# B&R Automation Studio project perfxxl (part 11)

#### rinse.c
```c
#ifdef _DEFAULT_INCLUDES
	#include <AsDefault.h>
#endif
/*
                             *******************
******************************* C SOURCE FILE *******************************
**                           *******************                           **
**                                                                         **
** project  : BlueFin                                                      **
** filename : RINSE.C                                                      **
** version  : 1.11                                                         **
** date     : 20.11.2007                                                   **
**                                                                         **
*****************************************************************************
** Abstract                                                                **
** ========                                                                **
** Handling of rinse functions: Circulation, refill, replenishing,         **
** monitoring Level and (optional) circulation switch                      **
**                                                                         **
** Copyright (c) 2007, Krause-Biagosch GmbH                                **
** All rights reserved.                                                    **
**                                                                         **
*****************************************************************************
VERSION HISTORY:
----------------
Version     : 1.00
Date        : 06.03.2007
Revised by  : Herbert Aden
Description : Original version, moved functionality from
              developertank task to here.

Version     : 1.10
Date        : 03.05.2007
Revised by  : Herbert Aden
Description : added delay for Level not ok error and delays for
              level switch on and off signal

Version     : 1.11
Date        : 20.11.2007
Revised by  : Herbert Aden
Description : added flow control functionality in mode "freshwater only",
              requires the sensor to be mounted in the inflow tube
*/
#define _RINSE_C_SRC

/****************************************************************************/
/**                                                                        **/
/**                           INCLUDE FILES                                **/
/**                                                                        **/
/****************************************************************************/

#include "egmglob_var.h"

/****************************************************************************/
/**                                                                        **/
/**                       DEFINITIONS AND MACROS                           **/
/**                                                                        **/
/****************************************************************************/
/* NONE */

/****************************************************************************/
/**                                                                        **/
/**                      TYPEDEFS AND STRUCTURES                           **/
/**                                                                        **/
/****************************************************************************/
/* NONE */

/****************************************************************************/
/**                                                                        **/
/**                      PROTOTYPES OF LOCAL FUNCTIONS                     **/
/**                                                                        **/
/****************************************************************************/
/* NONE */

/****************************************************************************/
/**                                                                        **/
/**                      EXPORTED VARIABLES                                **/
/**                                                                        **/
/****************************************************************************/
/* NONE */

/****************************************************************************/
/**                                                                        **/
/**                           GLOBAL VARIABLES                             **/
/**                                                                        **/
/****************************************************************************/
/*NONE*/

/****************************************************************************/
/**                                                                        **/
/**                      TASK-LOCAL VARIABLES                              **/
/**                                                                        **/
/****************************************************************************/
_LOCAL    UINT                RinseValveTime,RinseValveTimeToGo;

/****************************************************************************/
/**                                                                        **/
/**                    MODULE-LOCAL VARIABLES                              **/
/**                                                                        **/
/****************************************************************************/
static    TP_10ms_typ         RinseReplenishmentValveTimer;

static    TON_10ms_typ        RinseLevelOKTimer,RinseLevelNOTOKTimer,
                              RinseLevelErrorTimer,
                              RinsePumpStartTimer,
                              RinseFlowDelay,
                              RinseRefillTimer,
                              RinsePumpOffTimer,
                              RefillValveSafetyTimer;

static    R_TRIGtyp           RinsePumpCmdR,
                              RinseValveCmdR,
                              LevelOKR,
                              LevelNOTOKR;
static    F_TRIGtyp           RinseValveCmdF;

static    UINT                TmpValveTimeRinse;
static    BOOL                RinseRefillActive;

/****************************************************************************/
/**                                                                        **/
/**                      EXTERNAL VARIABLES                                **/
/**                                                                        **/
/****************************************************************************/
extern BOOL	Pulse_1s;

/****************************************************************************/
/**                                                                        **/
/**                          EXPORTED FUNCTIONS                            **/
/**                                                                        **/
/****************************************************************************/
void Rinse(void);

/******************************************************************************/
void Rinse(void)
{
/*Level*/
	RinseLevelOKTimer.IN = EGMRinse.TankFull;
	RinseLevelOKTimer.PT = 500; /*5 sec*/
	TON_10ms(&RinseLevelOKTimer);

	RinseLevelNOTOKTimer.IN = !EGMRinse.TankFull;
	RinseLevelNOTOKTimer.PT = 500; /*5 sec*/
	TON_10ms(&RinseLevelNOTOKTimer);

	LevelOKR.CLK = RinseLevelOKTimer.Q;
	LevelNOTOKR.CLK = RinseLevelNOTOKTimer.Q;
	R_TRIG(&LevelOKR);
	R_TRIG(&LevelNOTOKR);
	if(LevelOKR.Q)
		EGMRinse.LevelNotInRange = FALSE;
	if(LevelNOTOKR.Q)
		EGMRinse.LevelNotInRange = TRUE;

/* Fehlermeldung verzögern, erst wird automatisch befüllt */
	RinseLevelErrorTimer.IN = EGMRinse.LevelNotInRange;
	RinseLevelErrorTimer.PT = 2000; /* 20 s */
	TON_10ms(&RinseLevelErrorTimer);
	EGM_AlarmBitField[4] = (ModulStatus_DI == 1) && RinseLevelErrorTimer.Q && (EGMRinseParam.ReplenishingMode != FRESHWATERONLY);

/* REPLENISHING Rinse*/
/* a) per plate*/
	if (Pulse_1s &&(CurrentState == S_PROCESSING)&& (EGMRinseParam.ReplenishingMode == REPLPERPLATE))
	{
		TmpValveTimeRinse =
				((RinseReplenishmentPlateCounter * EGMRinseParam.ReplenishmentPerPlate) / EGMRinseParam.PumpMlPerSec)*100;
		if (TmpValveTimeRinse >= EGMRinseParam.MinPumpOnTime)
		{
			RinseReplenishmentValveTimer.IN = 1;
			RinseReplenishmentPlateCounter = 0;
		}
	}

/* b) per area*/
	if (Pulse_1s &&(CurrentState == S_PROCESSING)&& (EGMRinseParam.ReplenishingMode == REPLPERSQM))
	{
		TmpValveTimeRinse =
				((RinseReplenishmentSqmCounter * EGMRinseParam.ReplenishmentPerSqm) / EGMRinseParam.PumpMlPerSec)*100;
		if (TmpValveTimeRinse >= EGMRinseParam.MinPumpOnTime)
		{
			RinseReplenishmentValveTimer.IN = 1;
			RinseReplenishmentSqmCounter = 0;
		}
	}

	if (EGMRinse.Valve != OPEN )
		RinseValveTime = TmpValveTimeRinse;

	if (RinseReplenishmentValveTimer.IN && (EGMRinse.Valve != OPEN ))
		RinseReplenishmentValveTimer.PT = RinseValveTime;

	if (EGMRinse.Valve == OPEN )
		RinseValveTimeToGo = RinseReplenishmentValveTimer.PT - RinseReplenishmentValveTimer.ET;
	else
		RinseValveTimeToGo = 0;

	TP_10ms(&RinseReplenishmentValveTimer);
	RinseReplenishmentValveTimer.IN = 0;

	RinseValveCmdR.CLK = RinseReplenishmentValveTimer.Q;
	R_TRIG(&RinseValveCmdR);
	if (RinseValveCmdR.Q && (EGMRinseParam.ReplenishingMode != FRESHWATERONLY))
		EGMRinse.Valve = OPEN;

/* Ventil zu nach Zeit oder wenn kein Automatik Modus*/
	RinseValveCmdF.CLK = RinseReplenishmentValveTimer.Q && EGMRinse.Auto;
	F_TRIG(&RinseValveCmdF);
	if ((RinseValveCmdF.Q && (EGMRinseParam.ReplenishingMode != FRESHWATERONLY)) || !ControlVoltageOk)
	{
		EGMRinse.Valve = CLOSE;
	}

/*Refill Rinse*/
	TON_10ms(&RinseRefillTimer);
/* automatisch befüllen nur, wenn nicht ausschliesslich Frischwasser verwendet wird*/
	if (EGMRinseParam.ReplenishingMode != FRESHWATERONLY)
	{
		RinseRefillTimer.IN = !EGMRinse.LevelNotInRange;
		RinseRefillTimer.PT = 200;
/* Füllen nur wenn Automatik modus*/
		if (EGMRinse.LevelNotInRange && ControlVoltageOk && EGMRinse.Auto)
		{
			RinseRefillActive = TRUE;
			EGMRinse.Valve = OPEN;
		}
		if ((RinseRefillTimer.Q || !EGMRinse.Auto) && RinseRefillActive)
		{
			RinseRefillActive = FALSE;
			EGMRinse.Valve = CLOSE;
		}
	}
	else
	{
		RinseRefillTimer.IN = 0;
		RinseRefillActive = FALSE;
	}

/*
 * safety: if Valve is open and Tank full indicated close the valve after 10 sec
 */
	RefillValveSafetyTimer.IN = (EGMRinse.Valve == OPEN) && EGMRinse.TankFull;
	RefillValveSafetyTimer.PT = 1000; /* 10 sec */
	TON_10ms(&RefillValveSafetyTimer);

	if(RefillValveSafetyTimer.Q)
		EGMRinse.Valve = CLOSE;

/*Rinse Pump*/
	RinsePumpCmdR.CLK = EGMRinse.PumpCmd;
	R_TRIG(&RinsePumpCmdR);

/****************************************************************************/
/**                          Flow control                                  **/
/****************************************************************************/
	if(	EGMGlobalParam.UseRinseFlowControl )
	{
	/*
	 * wenn ausschliesslich Frischwasser verwendet wird,
	 * dann darf flow control nur  auf das geöffnete Ventil reagieren
	 */
		if (EGMRinseParam.ReplenishingMode == FRESHWATERONLY)
		{
		/*
		 * 20 sec nach Öffnen muss Durchfluß da sein
		 */
			RinsePumpStartTimer.IN = EGMRinse.Valve;
			RinsePumpStartTimer.PT = 2000; /* 20 sec */
			TON_10ms(&RinsePumpStartTimer);
			if( RinsePumpStartTimer.Q && !RinseFlowInput )
				EGM_AlarmBitField[36] = TRUE;
		}
		else
		{
	/*
	 * 20 sec nach Start der Pumpe muss Durchfluß da sein
	 */
			RinsePumpStartTimer.IN = EGMRinse.Pump;
			RinsePumpStartTimer.PT = 2000; /* 20 sec */
			TON_10ms(&RinsePumpStartTimer);
	/*
	 * wenn Frischwasser zugeführt wird, schaltet der Durchflußwächter ab,
	 * deshalb hier die Verriegelung des Fehlers mit dem Ventil
	 */
			RinseFlowDelay.IN = !RinseFlowInput && !EGMRinse.Valve;
			RinseFlowDelay.PT = 300; /* 3 sec */
			TON_10ms(&RinseFlowDelay);
			if( RinsePumpStartTimer.Q && RinseFlowDelay.Q )
				EGM_AlarmBitField[36] = TRUE;
		}
	}
	else
		EGM_AlarmBitField[36] = FALSE;

/* Rinse Pump
 * wenn 30 sec der Level nicht ok war wird die Pumpe abgeschaltet.
 * Sie kann durch steigende Flanke des Kommandos wieder für 30 s eingeschaltet werden
 * (für Service)
*/
	RinsePumpOffTimer.IN = EGMRinse.LevelNotInRange && !RinsePumpCmdR.Q;
	RinsePumpOffTimer.PT = 3000; /*30 sec*/
	TON_10ms(&RinsePumpOffTimer);
	if (RinsePumpOffTimer.Q || !ControlVoltageOk || EGM_AlarmBitField[36])
	{
		EGMRinse.Pump = OFF;
		EGMRinse.PumpCmd = OFF;
	}
	else
		EGMRinse.Pump = EGMRinse.PumpCmd;

}
/****************************************************************************/
/**                                                                        **/
/**                                 EOF                                    **/
/**                                                                        **/
/****************************************************************************/
```

#### gum.c
```c
#ifdef _DEFAULT_INCLUDES
	#include <AsDefault.h>
#endif
/*
                             *******************
******************************* C SOURCE FILE *******************************
**                           *******************                           **
**                                                                         **
** project  : BlueFin                                                      **
** filename : GUM.C                                                        **
** version  : 1.12                                                         **
** date     : 21.11.2007                                                   **
**                                                                         **
*****************************************************************************
** Abstract                                                                **
** ========                                                                **
** Handling of gumming functions: Circulation, monitoring Level            **
** and (optional) circulation switch                                       **
**                                                                         **
** Copyright (c) 2007, Krause-Biagosch GmbH                                **
** All rights reserved.                                                    **
**                                                                         **
*****************************************************************************
VERSION HISTORY:
----------------
Version     : 1.00
Date        : 06.03.2007
Revised by  : Herbert Aden
Description : Original version, moved functionality from
              developertank task to here.

Version     : 1.11
Date        : 16.11.2007
Revised by  : Herbert Aden
Description : added checking for gum valve output by monitoring an input

Version     : 1.12
Date        : 21.11.2007
Revised by  : Herbert Aden
Description : removed checking for gum valve output by monitoring an input
              (was for testing at Bauer only)
*/
#define _GUM_C_SRC

/****************************************************************************/
/**                                                                        **/
/**                           INCLUDE FILES                                **/
/**                                                                        **/
/****************************************************************************/

#include "egmglob_var.h"

/****************************************************************************/
/**                                                                        **/
/**                       DEFINITIONS AND MACROS                           **/
/**                                                                        **/
/****************************************************************************/
/* NONE */

/****************************************************************************/
/**                                                                        **/
/**                      TYPEDEFS AND STRUCTURES                           **/
/**                                                                        **/
/****************************************************************************/
/* NONE */

/****************************************************************************/
/**                                                                        **/
/**                      PROTOTYPES OF LOCAL FUNCTIONS                     **/
/**                                                                        **/
/****************************************************************************/
/* NONE */

/****************************************************************************/
/**                                                                        **/
/**                      EXPORTED VARIABLES                                **/
/**                                                                        **/
/****************************************************************************/
/* NONE */

/****************************************************************************/
/**                                                                        **/
/**                           GLOBAL VARIABLES                             **/
/**                                                                        **/
/****************************************************************************/
/*NONE*/

/****************************************************************************/
/**                                                                        **/
/**                      TASK-LOCAL VARIABLES                              **/
/**                                                                        **/
/****************************************************************************/
/*NONE*/

/****************************************************************************/
/**                                                                        **/
/**                    MODULE-LOCAL VARIABLES                              **/
/**                                                                        **/
/****************************************************************************/
static    TON_10ms_typ        GumLevelTimer,GumFlowingDelay;
static    TON_10ms_typ        GumPumpOffTimer,GumPumpStartTimer;

static    R_TRIGtyp           GumPumpCmdR;

/****************************************************************************/
/**                                                                        **/
/**                      EXTERNAL VARIABLES                                **/
/**                                                                        **/
/****************************************************************************/
extern BOOL	Pulse_1s;

/****************************************************************************/
/**                                                                        **/
/**                          EXPORTED FUNCTIONS                            **/
/**                                                                        **/
/****************************************************************************/
void Gum(void);
void InitGum(void);

/******************************************************************************/
void InitGum(void)
{
	return;
}

/******************************************************************************/
void Gum(void)
{

	if(!EGMGlobalParam.EnableGumSection && (MachineType != BLUEFIN_XS))
	{
		EGM_AlarmBitField[2] = FALSE;
		EGM_AlarmBitField[33] = FALSE;
		EGMGum.LevelNotInRange = FALSE;
		EGMGum.Pump = OFF;
		EGMGum.PumpCmd = OFF;
		EGMGum.Valve = OFF;
		EGMGum.RinseValve = OFF;
		return;
	}

/*Level Gum*/
	GumLevelTimer.IN = !EGMGum.TankFull;
	GumLevelTimer.PT = 200; /*2 sec*/
	TON_10ms(&GumLevelTimer);
	EGMGum.LevelNotInRange = GumLevelTimer.Q;
	EGM_AlarmBitField[2] = (ModulStatus_DI == 1) && EGMGum.LevelNotInRange;
/*Gum Pump*/
	GumPumpCmdR.CLK = EGMGum.PumpCmd;
	R_TRIG(&GumPumpCmdR);

	if(	EGMGlobalParam.UseGumFlowControl )
	{
	/* flow control starts 20 sec after pump start */
		GumPumpStartTimer.IN = EGMGum.Pump;
		GumPumpStartTimer.PT = 2000; /*20 sec*/
		TON_10ms(&GumPumpStartTimer);

	/* delay the "not flowing" error a bit */
		GumFlowingDelay.IN = !GumFC.Flowing;
		GumFlowingDelay.PT = 300; /* 3sec */
		TON_10ms(&GumFlowingDelay);

		if( GumPumpStartTimer.Q && GumFlowingDelay.Q )
		{
			EGM_AlarmBitField[33] = TRUE;
			GumFC.ResetMlFlown = TRUE;
		}
	}
	else
		EGM_AlarmBitField[33] = FALSE;

/* manual retrigger of the pump is possible, it will run for 5 sec */
	GumPumpOffTimer.IN = EGMGum.LevelNotInRange && !GumPumpCmdR.Q;
	GumPumpOffTimer.PT = 500; /*5 sec*/
	TON_10ms(&GumPumpOffTimer);
	if (GumPumpOffTimer.Q || !ControlVoltageOk || EGM_AlarmBitField[33])
	{
		EGMGum.Pump = OFF;
		EGMGum.PumpCmd = OFF;
	}
	else
		EGMGum.Pump = EGMGum.PumpCmd;

/*
 * safety: if the gum pump is running we always want the gum valve switched
 * and the Rinse valve closed
 */
	if( EGMGum.Pump )
	{
		EGMGum.Valve = ON;
		EGMGum.RinseValve = CLOSE;
	}

/*
 * safety: if gum rinse valve is switched on, then
 * we always want the gum valve to be switched off to make sure the
 * rinsing water cannot flow into the gum tank;
 * the Pump is switched off as well
 */
	if( EGMGum.RinseValve == OPEN )
	{
		EGMGum.Pump = EGMGum.PumpCmd = OFF;
		EGMGum.Valve = OFF;
	}
}
/****************************************************************************/
/**                                                                        **/
/**                                 EOF                                    **/
/**                                                                        **/
/****************************************************************************/
```

#### tanks.c
```c
#ifdef _DEFAULT_INCLUDES
	#include <AsDefault.h>
#endif
/*
                             *******************
******************************* C SOURCE FILE *******************************
**                           *******************                           **
**                                                                         **
** project  : BlueFin                                                      **
** filename : TANKS.C                                                      **
** version  : 1.10                                                         **
** date     : 09.03.2007                                                   **
**                                                                         **
*****************************************************************************
** Abstract                                                                **
** ========                                                                **
** Handling of Prewash, Rinse and Gum stations, basically just call        **
** functions of respective source files                                    **
**                                                                         **
** Copyright (c) 2007, Krause-Biagosch GmbH                                **
** All rights reserved.                                                    **
**                                                                         **
*****************************************************************************
VERSION HISTORY:
----------------
Version     : 1.00
Date        : 06.03.2007
Revised by  : Herbert Aden
Description : Original version, moved functionality from
              developertank task to here.

Version     : 1.10
Date        : 03.05.2007
Revised by  : Herbert Aden
Description : changes in rinse.c and prewash.c
*/
#define _TANKS_C_SRC

/****************************************************************************/
/**                                                                        **/
/**                           INCLUDE FILES                                **/
/**                                                                        **/
/****************************************************************************/
#include "egmglob_var.h"

/****************************************************************************/
/**                                                                        **/
/**                       DEFINITIONS AND MACROS                           **/
/**                                                                        **/
/****************************************************************************/
/* NONE */

/****************************************************************************/
/**                                                                        **/
/**                      TYPEDEFS AND STRUCTURES                           **/
/**                                                                        **/
/****************************************************************************/
/* NONE */

/****************************************************************************/
/**                                                                        **/
/**                      PROTOTYPES OF LOCAL FUNCTIONS                     **/
/**                                                                        **/
/****************************************************************************/
/* NONE */

/****************************************************************************/
/**                                                                        **/
/**                      PRTOTYPES OF EXTERNAL FUNCTIONS                   **/
/**                                                                        **/
/****************************************************************************/
extern void Prewash(void);
extern void Rinse(void);
extern void Gum(void);
extern void InitGum(void);

/****************************************************************************/
/**                                                                        **/
/**                      EXPORTED VARIABLES                                **/
/**                                                                        **/
/****************************************************************************/
/* NONE */

/****************************************************************************/
/**                                                                        **/
/**                           GLOBAL VARIABLES                             **/
/**                                                                        **/
/****************************************************************************/
/*NONE*/

/****************************************************************************/
/**                                                                        **/
/**                      TASK-LOCAL VARIABLES                              **/
/**                                                                        **/
/****************************************************************************/
/*NONE*/

/****************************************************************************/
/**                                                                        **/
/**                    MODULE-LOCAL VARIABLES                              **/
/**                                                                        **/
/****************************************************************************/
static    TON_10ms_typ        PulseTimer1;

/****************************************************************************/
/**                                                                        **/
/**                      EXPORTED VARIABLES                                **/
/**                                                                        **/
/****************************************************************************/
BOOL	Pulse_1s;

/****************************************************************************/
/**                                                                        **/
/**                          LOCAL FUNCTIONS                               **/
/**                                                                        **/
/****************************************************************************/

/****************************************************************************/
/** Init function, executed once at startup                                **/
/****************************************************************************/
_INIT void init()
{
	PulseTimer1.IN = 0;
	PulseTimer1.PT = 100;
	InitGum();
}

/****************************************************************************/
/** Cyclic function                                                        **/
/****************************************************************************/
_CYCLIC void cyclic()
{

	PulseTimer1.IN = 1;
	if(PulseTimer1.Q)
		PulseTimer1.IN = 0;
	TON_10ms(&PulseTimer1);
	Pulse_1s = PulseTimer1.Q;

	if(MachineType == BLUEFIN_XS)
	{
		Prewash();
		Rinse();
	}

	Gum();
	return;
}
/****************************************************************************/
/**                                                                        **/
/**                                 EOF                                    **/
/**                                                                        **/
/****************************************************************************/
```

### Program Logical/ping (ANSIC)

#### ping.c - Zyklischer Code
```c
#ifdef _DEFAULT_INCLUDES
	#include <AsDefault.h>
#endif
/****************************************************************************/
/*	TCP/IP Client Funktionalität 											*/
/*																			*/
/*																			*/
/*	Versionsgeschichte:														*/
/*  Version		Datum		Änderung								von		*/
/*	1.0			25.02.03	erste Implementation der				HA		*/
/*							Ping Funktion									*/
/*	1.10		26.02.03	SMTP Client								HA		*/
/*	1.11		15.10.15	SMTP Client removed						HA		*/
/*																			*/
/****************************************************************************/

/***** Include-Files: *****/
#include <bur/plc.h>
#include <bur/plctypes.h>
#include <string.h>
/* damit das switch unten funktioniert*/
#define _REPLACE_CONST
#include <AsICMP.h>
#include "glob_var.h"
#include <AsBrStr.h>

/***** Variablen-/Konstantendeklaration: *****/

#ifndef TRUE
#define TRUE				1
#endif
#ifndef FALSE
#define FALSE				0
#endif

USINT PingOK,PingError;
_LOCAL	IcmpPing_typ PingVar;
_LOCAL	UINT	PingOKInvisible,PingErrorInvisible;
_LOCAL USINT StartPing,IPAdr1,IPAdr2,IPAdr3,IPAdr4;

STRING IPAdress[16],tmp[10];
TOF_10ms_typ PingLEDOff;

void Ping(void)
{
	PingOKInvisible = !PingOK;
	PingErrorInvisible = !PingError;
	PingLEDOff.IN = StartPing;
	PingLEDOff.PT = 300;
	TOF_10ms(&PingLEDOff);
	if(!PingLEDOff.Q)
	{
		PingOK = 0;
		PingError = 0;
	}
	if(StartPing)
	{
		PingVar.enable = TRUE;			/* FUB enable */
		strcpy(IPAdress,"");
		brsitoa(IPAdr1,(UDINT) &tmp[0]);
		strcat(IPAdress,tmp);
		strcat(IPAdress,".");
		brsitoa(IPAdr2,(UDINT) &tmp[0]);
		strcat(IPAdress,tmp);
		strcat(IPAdress,".");
		brsitoa(IPAdr3,(UDINT) &tmp[0]);
		strcat(IPAdress,tmp);
		strcat(IPAdress,".");
		brsitoa(IPAdr4,(UDINT) &tmp[0]);
		strcat(IPAdress,tmp);
		PingVar.pHost = (UDINT)IPAdress;	/* IP Address of the Reciever */
		PingVar.timeout = 100;			/* Time of waiting */
		PingOK = 0;
		PingError = 0;
		IcmpPing(&PingVar);
		switch(PingVar.status)
		{
			case ERR_OK:
			{
				/* Ping OK */
				StartPing = FALSE;
				PingOK = 1;
				PingError = 0;
				/***********************/
				/* TODO: Go on working */
				/***********************/
				break;
			}
			case ERR_FUB_BUSY:
				/* Fub is already working */
				/* call again */
				break;
			case icmpERR_NO_RESPONSE:
			{
				/* No Response */
				/*************************/
				/* TODO: Failure routine */
				/*************************/
				StartPing = FALSE;
				PingError = 1;
				PingOK = 0;
				break;
			}
			case icmpERR_PARAMETER:
			case icmpERR_SOCKET_CREATE:
			case icmpERR_SYSTEM:
			{
				/* Response timedout */
				/***************************/
				/* TODO: Failure routine   */
				/*		 Timeout to short? */
				/***************************/
				StartPing = FALSE;
				PingError = 1;
				PingOK = 0;
				break;
			}
			default:
			{
				/* Error occurs */
				StartPing = FALSE;
				/*************************/
				/* TODO: Failure routine */
				/*************************/
				PingError = 1;
				PingOK = 0;
				break;
			}
		}
	}
}

/***** INIT FUNKTION *******************************************************/
_INIT void init (void)
{
	IPAdr1 = 192;
	IPAdr2 = 168;
	IPAdr3 = 77;
	IPAdr4 = 99;
} /* Ende Funktion _INIT void init (void) */

/***** ZYKLISCHE FUNKTION **************************************************/
_CYCLIC void cyclic (void)
{
	Ping();

} /* Ende Funktion _CYCLIC void cyclic (void) */

/* ENDE */
```

Listed in the project but not available here: Logical/file/auxfunc.c, Logical/hwconfig/auxfunc.c, Logical/udp_nl/auxfunc.c, Logical/Exposer/Hardware/motoren/motorfunc.c, Logical/Exposer/Ablauf/referenz/auxfunc.c, Logical/Exposer/Ablauf/entladen/auxfunc.c, Logical/Exposer/Ablauf/adjust/motorfunc.c, Logical/Exposer/Ablauf/adjust/auxfunc.c, Logical/Exposer/Ablauf/aufnahme/motorfunc.c, Logical/Exposer/Ablauf/aufnahme/auxfunc.c, Logical/Processor/preheat/auxfunc.c, Logical/Processor/devtank/auxfunc.c, Logical/Processor/egmauto/auxfunc.c
